PROGRAM MAIN
VAR
	//Stati
	IN_FUNZIONE: BOOL;
	IN_SIGILLATURA: BOOL;
	IN_SMISTAMENTO: BOOL;
	SCATOLA_ALTA: BOOL;
	SCATOLA_BASSA: BOOL;
	
	//Timer
	TON_SIGILLATURA: TON;
	TON_RILEVAZIONE_ALTEZZA: TON;
	TON_SMISTAMENTO_ALTI: TON;

	//Counter
	CTU_ALTI: CTU;
	CTU_BASSI: CTU;
	STOP_CONFERMATO: BOOL;
	STOP_RICHIESTO: BOOL;
	TON_STOP: TON;
	IN_ANOMALIA: BOOL;
	TON_ANOMALIA: TON;
	CONTROLLO_ALTEZZA: BOOL;
	TON_ANOMALIA_ALTEZZA: TON;
	IN_RILEVAZIONE_ALTEZZA: BOOL;
	TON_FINECORSA_SIGILLATURA: TON;
	RILASCIA_PISTONE: BOOL;
END_VAR

GestioneAnomalie();
GestioneStop();
GestionePulsantiSegnalazioni();
GestioneMotori();
GestioneSigillatura();
GestioneSmistamento();
GestioneConteggio();

ACTION GestioneAnomalie:
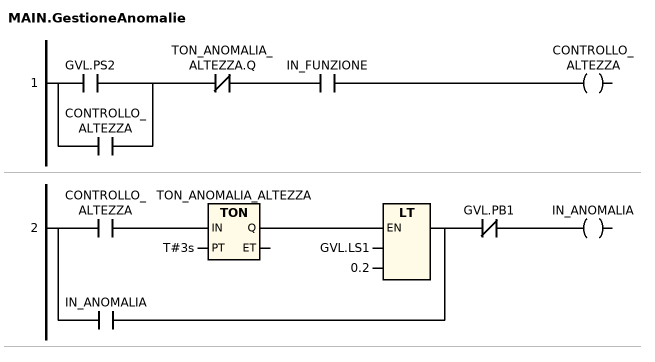
// NETWORK 1
CONTROLLO_ALTEZZA := (GVL.PS2 OR CONTROLLO_ALTEZZA) AND NOT TON_ANOMALIA_ALTEZZA.Q AND IN_FUNZIONE;

// NETWORK 2
TON_ANOMALIA_ALTEZZA(IN := CONTROLLO_ALTEZZA, PT := T#3s); // TON
IN_ANOMALIA := (TON_ANOMALIA_ALTEZZA.Q AND GVL.LS1 < 0.2 OR IN_ANOMALIA) AND NOT GVL.PB1;
END_ACTION

ACTION GestioneConteggio:
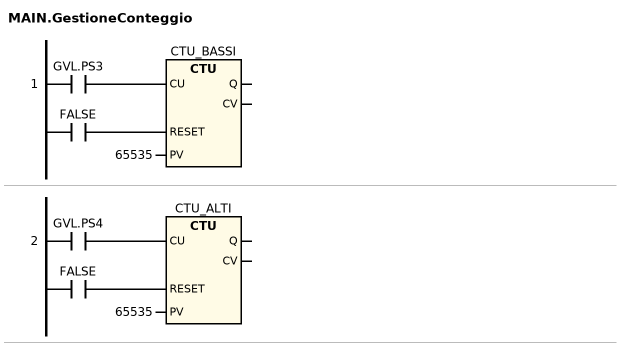
// NETWORK 1
CTU_BASSI(CU := GVL.PS3, RESET := FALSE, PV := 65535); // CTU

// NETWORK 2
CTU_ALTI(CU := GVL.PS4, RESET := FALSE, PV := 65535); // CTU
END_ACTION

ACTION GestioneMotori:
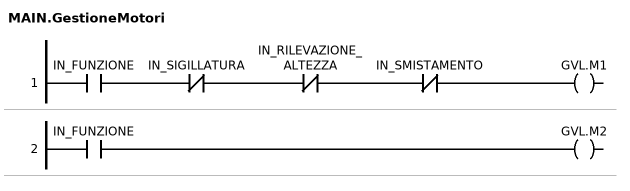
// NETWORK 1
GVL.M1 := IN_FUNZIONE AND NOT IN_SIGILLATURA AND NOT IN_RILEVAZIONE_ALTEZZA AND NOT IN_SMISTAMENTO;

// NETWORK 2
GVL.M2 := IN_FUNZIONE;
END_ACTION

ACTION GestionePulsantiSegnalazioni:
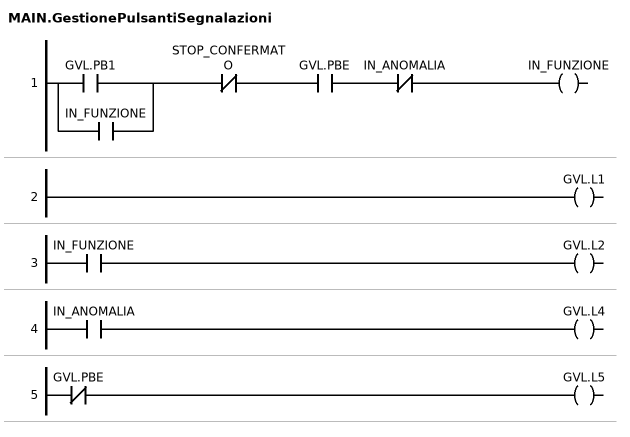
// NETWORK 1
IN_FUNZIONE := (GVL.PB1 OR IN_FUNZIONE) AND NOT STOP_CONFERMATO AND GVL.PBE AND NOT IN_ANOMALIA;

// NETWORK 2
GVL.L1 := TRUE;

// NETWORK 3
GVL.L2 := IN_FUNZIONE;

// NETWORK 4
GVL.L4 := IN_ANOMALIA;

// NETWORK 5
GVL.L5 := NOT GVL.PBE;
END_ACTION

ACTION GestioneSigillatura:
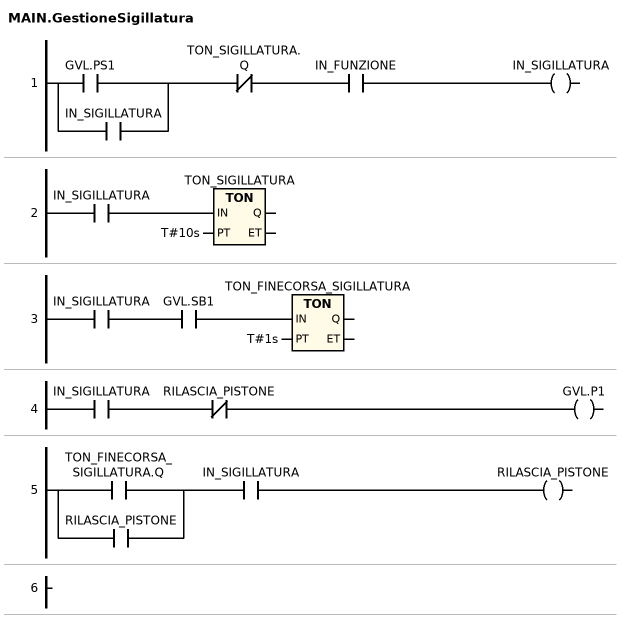
// NETWORK 1
IN_SIGILLATURA := (GVL.PS1 OR IN_SIGILLATURA) AND NOT TON_SIGILLATURA.Q AND IN_FUNZIONE;

// NETWORK 2
TON_SIGILLATURA(IN := IN_SIGILLATURA, PT := T#10s); // TON

// NETWORK 3
TON_FINECORSA_SIGILLATURA(IN := IN_SIGILLATURA AND GVL.SB1, PT := T#1s); // TON

// NETWORK 4
GVL.P1 := IN_SIGILLATURA AND NOT RILASCIA_PISTONE;

// NETWORK 5
RILASCIA_PISTONE := (TON_FINECORSA_SIGILLATURA.Q OR RILASCIA_PISTONE) AND IN_SIGILLATURA;

// NETWORK 6
END_ACTION

ACTION GestioneSmistamento:
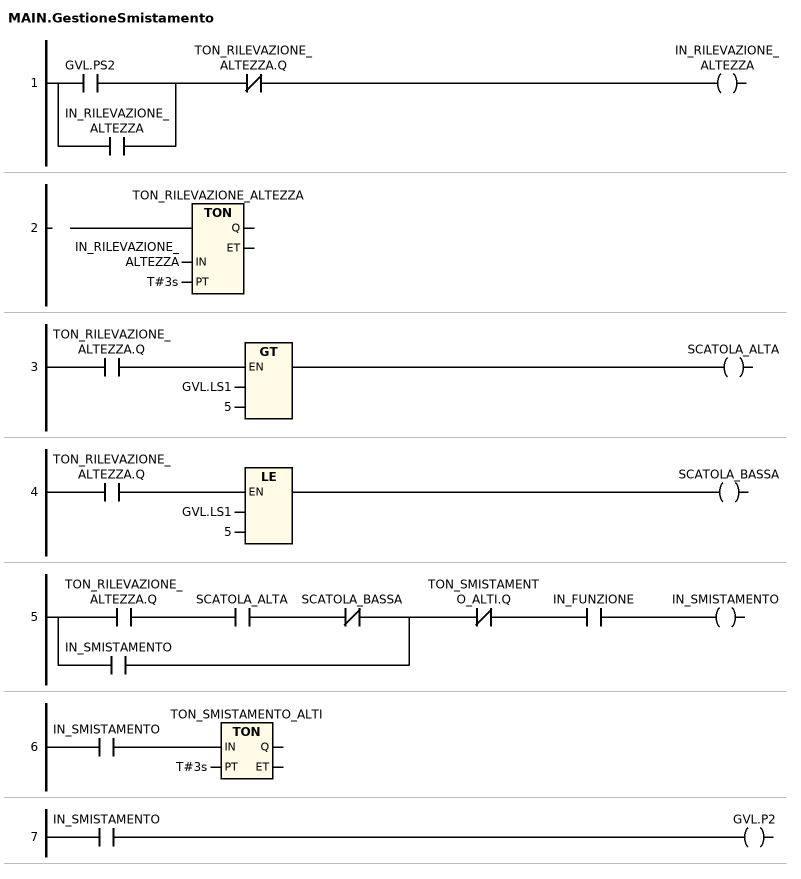
// NETWORK 1
IN_RILEVAZIONE_ALTEZZA := (GVL.PS2 OR IN_RILEVAZIONE_ALTEZZA) AND NOT TON_RILEVAZIONE_ALTEZZA.Q;

// NETWORK 2
TON_RILEVAZIONE_ALTEZZA(IN := IN_RILEVAZIONE_ALTEZZA, PT := T#3s); // TON

// NETWORK 3
SCATOLA_ALTA := TON_RILEVAZIONE_ALTEZZA.Q AND GVL.LS1 > 5;

// NETWORK 4
SCATOLA_BASSA := TON_RILEVAZIONE_ALTEZZA.Q AND GVL.LS1 <= 5;

// NETWORK 5
IN_SMISTAMENTO := (TON_RILEVAZIONE_ALTEZZA.Q AND SCATOLA_ALTA AND NOT SCATOLA_BASSA OR IN_SMISTAMENTO) AND NOT TON_SMISTAMENTO_ALTI.Q AND IN_FUNZIONE;

// NETWORK 6
TON_SMISTAMENTO_ALTI(IN := IN_SMISTAMENTO, PT := T#3s); // TON

// NETWORK 7
GVL.P2 := IN_SMISTAMENTO;
END_ACTION

ACTION GestioneStop:
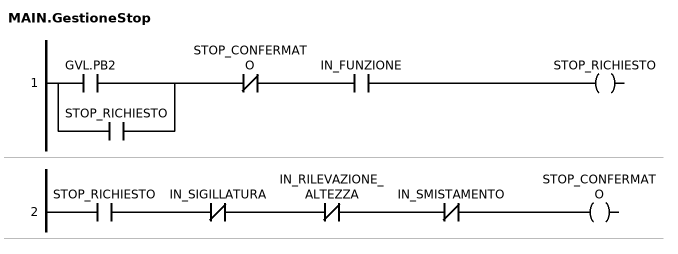
// NETWORK 1
STOP_RICHIESTO := (GVL.PB2 OR STOP_RICHIESTO) AND NOT STOP_CONFERMATO AND IN_FUNZIONE;

// NETWORK 2
STOP_CONFERMATO := STOP_RICHIESTO AND NOT IN_SIGILLATURA AND NOT IN_RILEVAZIONE_ALTEZZA AND NOT IN_SMISTAMENTO;
END_ACTION

END_PROGRAM

(* stored: Version 1.1.0.1, ProductVersion 3.1.4024.12
   POU MAIN: Id {77ce3c58-9155-42f5-9eb6-c02febfddbf9}, SpecialFunc None
   Action GestioneAnomalie: Id {81b64071-01a5-49a4-8a9c-d1881a4ec06b}
   Action GestioneConteggio: Id {619b20d3-e452-44f5-b626-dfa96b8409ac}
   Action GestioneMotori: Id {9e464890-6681-41a5-8f39-3082d5bac0ef}
   Action GestionePulsantiSegnalazioni: Id {3f00a759-f8d0-455e-af78-03f29b3994ec}
   Action GestioneSigillatura: Id {1a6fd54d-5c27-49f7-a49b-40229ed8561a}
   Action GestioneSmistamento: Id {6f07de2f-68ba-41e8-a08f-d2eacd4f38eb}
   Action GestioneStop: Id {dd2056fa-1f28-46ea-955b-d265caa7f59a} *)
